{attribute 'GeneratedUsingTerminal: EPP2316-0003-0016'}
{attribute addProperty BoxType "EPP2316-0003-0016"}
{attribute addProperty Id "EtcSlaveTerminalBaseDIG_InputsAT %I*DIG_Inputs_CC4551489DIG_Diag_InputsAT %I*DIG_Diag_Inputs_584303BF8DIG_Inputs_DeviceAT %I*DIG_Inputs_Device_E94E5BF95DIG_OutputsAT %Q*DIG_Outputs_28AC1A9E8DIG_Outputs_DeviceAT %Q*DIG_Outputs_Device_36A5EF172WcStateAT %I*WcState_9091E0EB2InfoDataAT %I*InfoData_32EB74EA10"}
{attribute addProperty CRC "2897566935"}
{attribute addProperty Size "44"}
TYPE EPP2316_ACB55CD7 EXTENDS EtcSlaveTerminalBase :
STRUCT
	{attribute addProperty Name "DIG_Inputs"}
	DIG_Inputs : DIG_Inputs_CC455148;
	{attribute addProperty Name "DIG_Diag_Inputs"}
	DIG_Diag_Inputs : DIG_Diag_Inputs_584303BF;
	{attribute addProperty Name "DIG_Inputs_Device"}
	DIG_Inputs_Device : DIG_Inputs_Device_E94E5BF9;
	{attribute addProperty Name "DIG_Outputs"}
	DIG_Outputs : DIG_Outputs_28AC1A9E;
	{attribute addProperty Name "DIG_Outputs_Device"}
	DIG_Outputs_Device : DIG_Outputs_Device_36A5EF17;
	{attribute addProperty Name "WcState"}
	WcState : WcState_9091E0EB;
	{attribute addProperty Name "InfoData"}
	InfoData : InfoData_32EB74EA;
END_STRUCT
END_TYPE

(* stored: Version 1.2.0.0, ProductVersion 3.1.4024.9
   DUT EPP2316_ACB55CD7: Id {daad26c5-f9bf-414f-bd26-4b3260e7746a} *)
